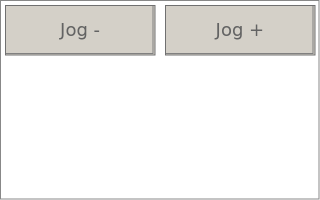
VISUALIZATION SingleAxisJogStandardSlow_1  // 320x200
VAR_IN_OUT
	btnJogPositive	: BOOL;
	btnJogNegative	: BOOL;
END_VAR
    Button (5,5 150x50), "Jog -"
        tap btnJogNegative
    Button (165,5 150x50), "Jog +"
        tap btnJogPositive
END_VISUALIZATION

(* stored: Version 1.1.0.1, ProductVersion 3.1.4024.12
   Visu SingleAxisJogStandardSlow_1: Id {30c2694b-4908-4186-8df2-73ae82f52afc} *)
